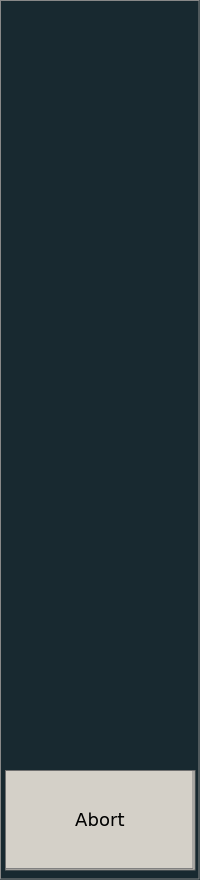
VISUALIZATION NavBarInitializing_1  // 200x880
VAR_IN_OUT
	btnAbort : BOOL;
END_VAR
    Button (5,770 190x100), "Abort"
        tap btnAbort
END_VISUALIZATION

(* stored: Version 1.1.0.1, ProductVersion 3.1.4024.12
   Visu NavBarInitializing_1: Id {446f2881-d9be-40a7-8cdb-e9b343d0dd89} *)
